TYPE ST_Interpreter_Inputs :
STRUCT
	
ZeroShiftDesc	: ZeroShiftDesc;

END_STRUCT
END_TYPE

(* stored: Version 1.1.0.1, ProductVersion 3.1.4024.9
   DUT ST_Interpreter_Inputs: Id {1c6ac9c5-002b-452e-aa05-6d7a79acb638} *)
